{attribute 'linkalways'} 
{attribute 'no_explicit_call' := 'This FB is a CLASS and must be accessed using methods or properties'}
{attribute 'enable_dynamic_creation'}
FUNCTION_BLOCK Node_F_VN_GetAt_TcVnKeyPoint EXTENDS VisionNode
VAR
    ipContainer : _ITcVnContainer;
    stElement : _TcVnKeyPoint;
    nIndex : _ULINT(0);
    hrPrev : _HRESULT(S_OK);
    hresult : _HRESULT(S_OK);
END_VAR

METHOD PUBLIC  Clone : I_Node
VAR
	pNode : POINTER TO Node_F_VN_GetAt_TcVnKeyPoint;
END_VAR
pNode := __NEW(Node_F_VN_GetAt_TcVnKeyPoint);
Clone := pNode^;
END_METHOD

METHOD FB_init : BOOL
VAR_INPUT
	bInitRetains : BOOL; // if TRUE, the retain variables are initialized (warm start / cold start)
	bInCopyCode : BOOL;  // if TRUE, the instance afterwards gets moved into the copy code (online change)
END_VAR
AddInput('ipContainer', ipContainer);
AddParameter('nIndex', nIndex);
AddInput('hrPrev', hrPrev);
AddOutput('stElement', stElement);
AddOutput('hresult',hresult);
END_METHOD

METHOD PROTECTED OnExecute
hresult.Value := F_VN_GetAt_TcVnKeyPoint(
    ipContainer := ipContainer.Value,
    stElement := stElement.Value,
    nIndex := nIndex.Value,
    hrPrev:= hrPrev.Value);
END_METHOD

METHOD PUBLIC PreExecutionCheck
VAR_INPUT
	Check : I_PreExecutionChecks;
END_VAR
Check.IsTrue(ipContainer.IsValid, 'ipContainer must be a valid container');
Check.IsTrue(ipContainer.IsType(TC_GLOBAL_CONST_LIST.ContainerType_Vector_TcVnKeyPoint), 'ipContainer contains incorrect type');
END_METHOD

END_FUNCTION_BLOCK

(* stored: Version 1.1.0.1, ProductVersion 3.1.4026.13
   POU Node_F_VN_GetAt_TcVnKeyPoint: Id {bd1f78df-62fc-4b53-a9b7-acaac5a0bf40}, SpecialFunc None
   Folder Constructor: Id {82319c66-ec82-4b3a-ae06-4bb93b17f7d7}
   Method Clone: Id {99b17620-56a7-4c5a-a407-e558c36e7a42}
   Method FB_init: Id {cb1bdedb-25a2-48b2-b8df-c08cda15fd3f}
   Method OnExecute: Id {1fd3268d-510b-45eb-be1f-7da19edf3866}
   Method PreExecutionCheck: Id {520ee026-b7ab-412b-b9d5-dae7eea64d90} *)
